TYPE ST_ReportControl :
STRUCT
	iIndex					:INT;
END_STRUCT
END_TYPE

(* stored: Version 1.1.0.1, ProductVersion 3.1.4024.12
   DUT ST_ReportControl: Id {1813ce86-f451-486c-a446-a38873298de1} *)
